FUNCTION_BLOCK Fb_Test_init_Cookie
VAR_INPUT
	execute: BOOL;
END_VAR

IF execute THEN
	MI5.Module2001.Input.SkillInput.SkillInput0.ParameterInput.ParameterInput0.StringValue := 'opc.tcp://192.168.192.136:4840';
	MI5.Module2001.Input.SkillInput.SkillInput0.ParameterInput.ParameterInput1.StringValue := 'MI5.Module2101.Output.PositionSensor';
	MI5.Module2001.Input.SkillInput.SkillInput0.ParameterInput.ParameterInput2.StringValue := 'MI5.Module2101.Input.PositionInput';
	MI5.Module2001.Input.SkillInput.SkillInput0.ParameterInput.ParameterInput3.StringValue := '4';
	MI5.Module2001.Input.SkillInput.SkillInput0.ParameterInput.ParameterInput4.StringValue := 'PLC1';
	MI5.Module2001.Input.SkillInput.SkillInput0.Execute := TRUE;
	IF MI5.Module2001.Output.SkillOutput.SkillOutput0.Done OR MI5.Module2001.Output.SkillOutput.SkillOutput0.Error THEN
		MI5.Module2001.Input.SkillInput.SkillInput0.Execute := FALSE;
		execute := FALSE;
	END_IF
END_IF

END_FUNCTION_BLOCK

(* stored: Version 1.1.0.1, ProductVersion 3.1.0.25
   POU Fb_Test_init_Cookie: Id {5eb876f7-2c6f-497d-b47a-dc79d3d86fde} *)
